{attribute addProperty BoxType "EP3204-0002-0017"}
{attribute addProperty Id "RTD_RTDInputs_ChannelAT %I*ARRAY[0..3] OF RTD_RTDInputs_Channel_4364CDB6296370WcStateAT %I*WcState_98A4DF7520.250InfoDataAT %I*InfoData_BC63D37F80100"}
{attribute addProperty CRC "271030498"}
{attribute addProperty SizeInBites "378"}
{attribute addProperty SizeInBytes "47.25"}
TYPE EP3204_72ABB954 :
STRUCT
	{attribute addProperty Name "RTD_RTDInputs_Channel"}
	RTD_RTDInputs_Channel : ARRAY[0..3] OF RTD_RTDInputs_Channel_4364CDB6;
	{attribute addProperty Name "WcState"}
	WcState : WcState_98A4DF75;
	{attribute addProperty Name "InfoData"}
	InfoData : InfoData_BC63D37F;
END_STRUCT
END_TYPE

(* stored: Version 1.2.0.0, ProductVersion 3.1.4024.9
   DUT EP3204_72ABB954: Id {07d4701f-a888-4f88-9d6b-4979d55f6af5} *)
